FUNCTION_BLOCK ForcibleBool_TEST
VAR
END_VAR

ForceOff();
ForceOn();
UnforcedOff();
UnforcedOn();

METHOD ForceOff
VAR
	Expected	 : BOOL;
	Actual		 : BOOL;
	ForcibleBool : ForcibleBool('');
END_VAR
IF TestSuite.Test(__POUNAME()).ExecuteTest() THEN
	Expected := FALSE;
	ForcibleBool.SetForceState(E_ForceState.ForceOff);
	ForcibleBool.Input := TRUE;
	Actual			   := ForcibleBool.Output;
	TestSuite.Test(__POUNAME()).AssertEqual(Expected, Actual);
END_IF
END_METHOD

METHOD ForceOn
VAR
	Expected	 : BOOL;
	Actual		 : BOOL;
	ForcibleBool : ForcibleBool('');
END_VAR
IF TestSuite.Test(__POUNAME()).ExecuteTest() THEN
	Expected := TRUE;
	ForcibleBool.SetForceState(E_ForceState.ForceOn);
	ForcibleBool.Input := FALSE;
	Actual			   := ForcibleBool.Output;
	TestSuite.Test(__POUNAME()).AssertEqual(Expected, Actual);
END_IF
END_METHOD

METHOD UnforcedOff
VAR
	Expected	 : BOOL;
	Actual		 : BOOL;
	ForcibleBool : ForcibleBool('');
END_VAR
IF TestSuite.Test(__POUNAME()).ExecuteTest() THEN
	Expected := FALSE;
	ForcibleBool.SetForceState(E_ForceState.Unforced);
	ForcibleBool.Input := FALSE;
	Actual			   := ForcibleBool.Output;
	TestSuite.Test(__POUNAME()).AssertEqual(Expected, Actual);
END_IF
END_METHOD

METHOD UnforcedOn
VAR
	Expected	 : BOOL;
	Actual		 : BOOL;
	ForcibleBool : ForcibleBool('');
END_VAR
IF TestSuite.Test(__POUNAME()).ExecuteTest() THEN
	Expected := TRUE;
	ForcibleBool.SetForceState(E_ForceState.Unforced);
	ForcibleBool.Input := TRUE;
	Actual			   := ForcibleBool.Output;
	TestSuite.Test(__POUNAME()).AssertEqual(Expected, Actual);
END_IF
END_METHOD

END_FUNCTION_BLOCK

(* stored: Version 1.1.0.1, ProductVersion 3.1.4026.18
   POU ForcibleBool_TEST: Id {fce2d78e-4523-495d-a99b-53d59e003270}, SpecialFunc None
   Method ForceOff: Id {88699ade-61bd-4059-a8a2-615a4cbf8a98}
   Method ForceOn: Id {004fb711-bf79-4a7b-a9f5-e5416fd7edf2}
   Method UnforcedOff: Id {329007b5-8123-45d1-882e-01c74a5fbc95}
   Method UnforcedOn: Id {4a1ed549-5c0b-456d-87a1-87bafdfa006b} *)
